FUNCTION_BLOCK M_MODBUSSLAVE
VAR_INPUT
END_VAR
VAR_OUTPUT
END_VAR
VAR
	_ENABLE : BOOL := FALSE;
	_FBSLAVE : ModbusRtuSlave_PcCOM;
	
	_MBINPUT 	: ARRAY[0..255] OF WORD;
	_MBOUTPUT 	: ARRAY[0..255] OF WORD;
	_MBMEMORY 	: ARRAY[0..255] OF WORD;
END_VAR

IF _ENABLE THEN
	_FBSLAVE(
		AdrInputs:= ADR(_MBINPUT), 
		SizeInputBytes:= SIZEOF(_MBINPUT), 
		AdrOutputs:= ADR(_MBOUTPUT), 
		SizeOutputBytes:= SIZEOF(_MBOUTPUT), 
		AdrMemory:= ADR(_MBMEMORY), 
		SizeMemoryBytes:= SIZEOF(_MBMEMORY), 
		ErrorId=> );
END_IF

PROPERTY ENABLE : BOOL
GET
ENABLE := _ENABLE;
END_GET
SET
_ENABLE := ENABLE;
END_SET
END_PROPERTY

METHOD FB_init : BOOL
VAR_INPUT
	bInitRetains : BOOL; // if TRUE, the retain variables are initialized (warm start / cold start)
	bInCopyCode : BOOL;  // if TRUE, the instance afterwards gets moved into the copy code (online change)

	DeviceID : UINT(1..247);
END_VAR
_FBSLAVE.UnitID := DeviceID;
END_METHOD

PROPERTY ID : UINT(1..247)
GET
ID := _FBSLAVE.UnitID;
END_GET
SET
_FBSLAVE.UnitID := ID;
END_SET
END_PROPERTY

PROPERTY INPUTS : POINTER TO BYTE
GET
INPUTS := ADR(_MBINPUT);
END_GET
END_PROPERTY

PROPERTY MEMORY : POINTER TO BYTE
GET
MEMORY := ADR(_MBMEMORY);
END_GET
END_PROPERTY

PROPERTY OUTPUTS : POINTER TO BYTE
GET
OUTPUTS := ADR(_MBOUTPUT);
END_GET
END_PROPERTY

END_FUNCTION_BLOCK

(* stored: Version 1.1.0.1, ProductVersion 3.1.4020.3
   POU M_MODBUSSLAVE: Id {223d5cf5-b74b-4cd8-b512-ae387b6f3c23}, SpecialFunc None
   Property ENABLE: Id {cef8f683-8592-44e2-97b8-8a48f73d8582}
   Get Get: Id {06745bcc-189f-4814-8b65-d72cbfcbd0ee}
   Set Set: Id {c4f01f8a-6a0f-4227-9644-a8ea21839e60}
   Method FB_init: Id {7c627f09-e8ec-417e-909f-705bb8db10e8}
   Property ID: Id {ddd00962-b084-4d3c-b23c-a99e977a4862}
   Get Get: Id {2c9d694a-4215-4e45-bb3a-b99e80303216}
   Set Set: Id {9a34f3ad-d965-43fe-97d8-aa9c60b81c79}
   Property INPUTS: Id {9a2041dd-2395-4579-b59b-b4506e5b8c4d}
   Get Get: Id {438cb3d1-aa45-4f4b-ae2a-1c33a949e524}
   Property MEMORY: Id {4fa84482-7b1e-49db-9453-e7c7cc215098}
   Get Get: Id {c1ee03c1-e3b4-409f-9df5-f21af0b6a2f2}
   Property OUTPUTS: Id {8d40b398-4c37-4d58-9bb3-01853b8def71}
   Get Get: Id {aea7b795-aa13-4964-a1ca-a75b62cec49b} *)
